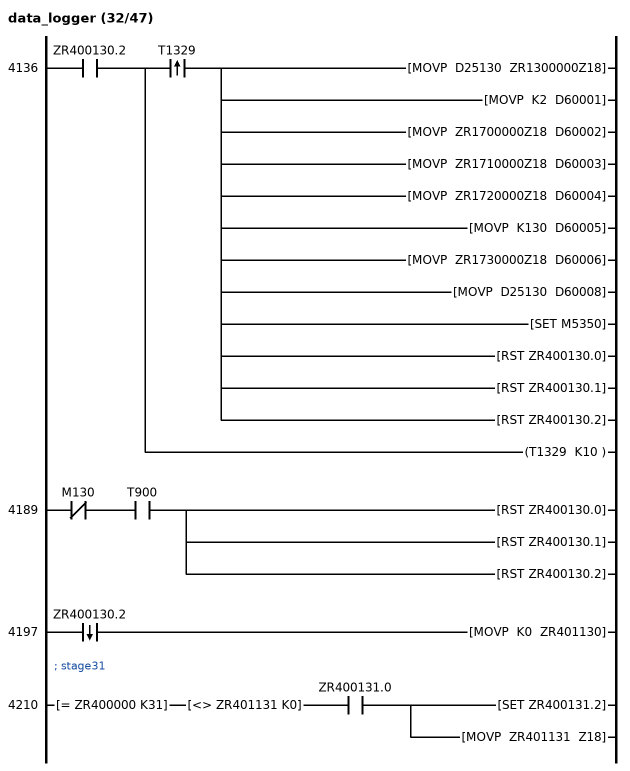
4136  LD      ZR400130.2
      MPS
      ANDP    T1329
      MOVP    D25130 ZR1300000Z18
      MOVP    K2 D60001
      MOVP    ZR1700000Z18 D60002
      MOVP    ZR1710000Z18 D60003
      MOVP    ZR1720000Z18 D60004
      MOVP    K130 D60005
      MOVP    ZR1730000Z18 D60006
      MOVP    D25130 D60008
      SET     M5350
      RST     ZR400130.0
      RST     ZR400130.1
      RST     ZR400130.2
      MPP
      OUT     T1329 K10
4189  LDI     M130
      AND     T900
      RST     ZR400130.0
      RST     ZR400130.1
      RST     ZR400130.2
4197  LDF     ZR400130.2
      MOVP    K0 ZR401130
; stage31
4210  LD=     ZR400000 K31
      AND<>   ZR401131 K0
      AND     ZR400131.0
      SET     ZR400131.2
      MOVP    ZR401131 Z18
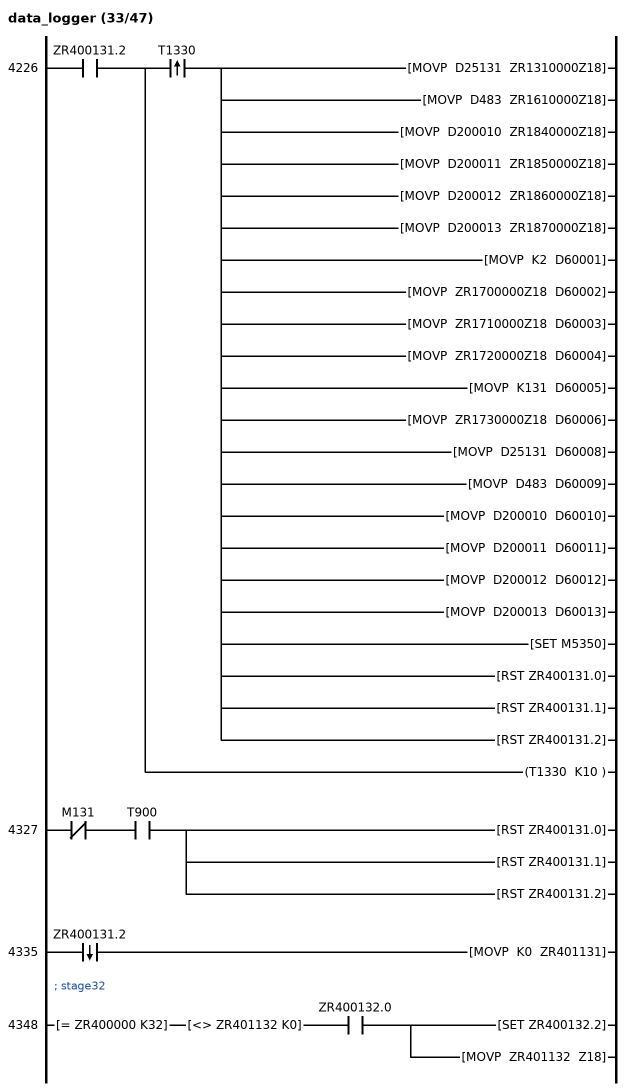
4226  LD      ZR400131.2
      MPS
      ANDP    T1330
      MOVP    D25131 ZR1310000Z18
      MOVP    D483 ZR1610000Z18
      MOVP    D200010 ZR1840000Z18
      MOVP    D200011 ZR1850000Z18
      MOVP    D200012 ZR1860000Z18
      MOVP    D200013 ZR1870000Z18
      MOVP    K2 D60001
      MOVP    ZR1700000Z18 D60002
      MOVP    ZR1710000Z18 D60003
      MOVP    ZR1720000Z18 D60004
      MOVP    K131 D60005
      MOVP    ZR1730000Z18 D60006
      MOVP    D25131 D60008
      MOVP    D483 D60009
      MOVP    D200010 D60010
      MOVP    D200011 D60011
      MOVP    D200012 D60012
      MOVP    D200013 D60013
      SET     M5350
      RST     ZR400131.0
      RST     ZR400131.1
      RST     ZR400131.2
      MPP
      OUT     T1330 K10
4327  LDI     M131
      AND     T900
      RST     ZR400131.0
      RST     ZR400131.1
      RST     ZR400131.2
4335  LDF     ZR400131.2
      MOVP    K0 ZR401131
; stage32
4348  LD=     ZR400000 K32
      AND<>   ZR401132 K0
      AND     ZR400132.0
      SET     ZR400132.2
      MOVP    ZR401132 Z18
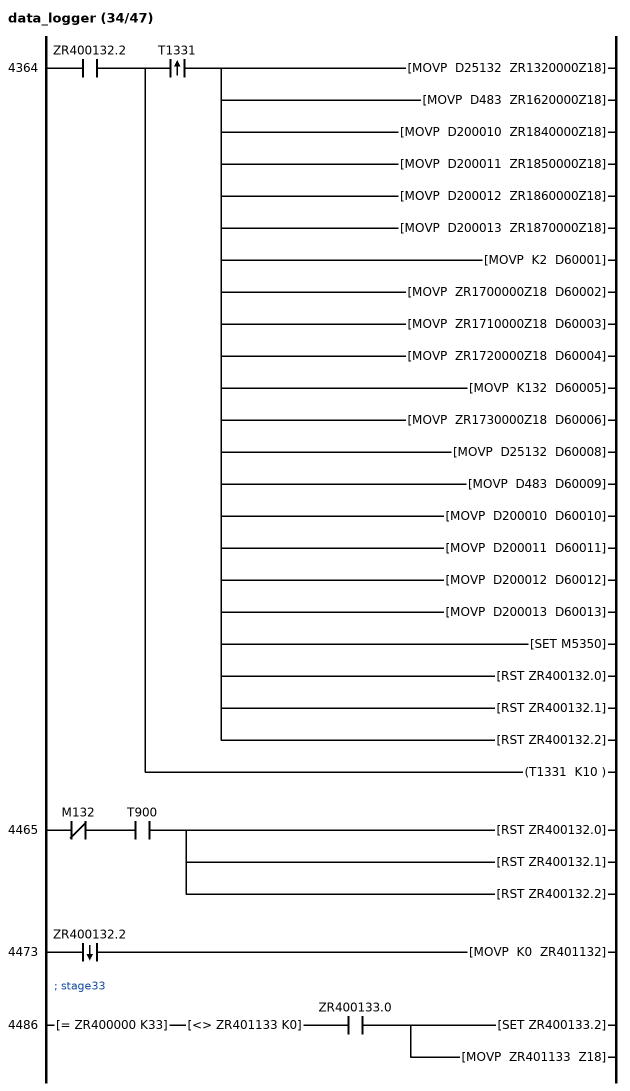
4364  LD      ZR400132.2
      MPS
      ANDP    T1331
      MOVP    D25132 ZR1320000Z18
      MOVP    D483 ZR1620000Z18
      MOVP    D200010 ZR1840000Z18
      MOVP    D200011 ZR1850000Z18
      MOVP    D200012 ZR1860000Z18
      MOVP    D200013 ZR1870000Z18
      MOVP    K2 D60001
      MOVP    ZR1700000Z18 D60002
      MOVP    ZR1710000Z18 D60003
      MOVP    ZR1720000Z18 D60004
      MOVP    K132 D60005
      MOVP    ZR1730000Z18 D60006
      MOVP    D25132 D60008
      MOVP    D483 D60009
      MOVP    D200010 D60010
      MOVP    D200011 D60011
      MOVP    D200012 D60012
      MOVP    D200013 D60013
      SET     M5350
      RST     ZR400132.0
      RST     ZR400132.1
      RST     ZR400132.2
      MPP
      OUT     T1331 K10
4465  LDI     M132
      AND     T900
      RST     ZR400132.0
      RST     ZR400132.1
      RST     ZR400132.2
4473  LDF     ZR400132.2
      MOVP    K0 ZR401132
; stage33
4486  LD=     ZR400000 K33
      AND<>   ZR401133 K0
      AND     ZR400133.0
      SET     ZR400133.2
      MOVP    ZR401133 Z18
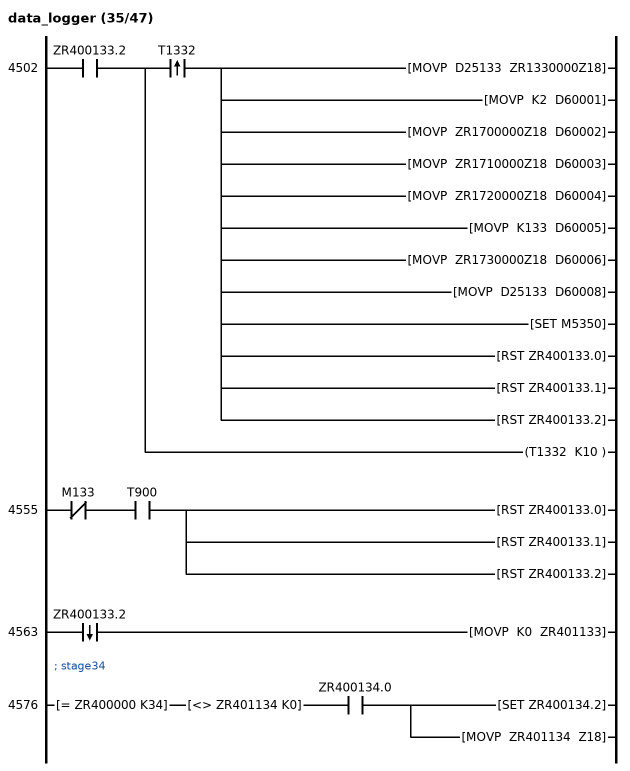
4502  LD      ZR400133.2
      MPS
      ANDP    T1332
      MOVP    D25133 ZR1330000Z18
      MOVP    K2 D60001
      MOVP    ZR1700000Z18 D60002
      MOVP    ZR1710000Z18 D60003
      MOVP    ZR1720000Z18 D60004
      MOVP    K133 D60005
      MOVP    ZR1730000Z18 D60006
      MOVP    D25133 D60008
      SET     M5350
      RST     ZR400133.0
      RST     ZR400133.1
      RST     ZR400133.2
      MPP
      OUT     T1332 K10
4555  LDI     M133
      AND     T900
      RST     ZR400133.0
      RST     ZR400133.1
      RST     ZR400133.2
4563  LDF     ZR400133.2
      MOVP    K0 ZR401133
; stage34
4576  LD=     ZR400000 K34
      AND<>   ZR401134 K0
      AND     ZR400134.0
      SET     ZR400134.2
      MOVP    ZR401134 Z18
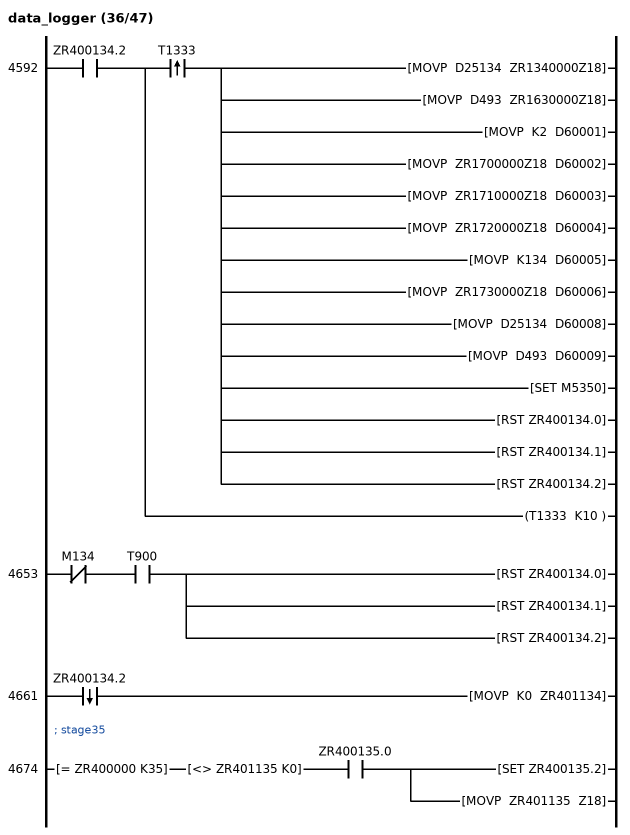
4592  LD      ZR400134.2
      MPS
      ANDP    T1333
      MOVP    D25134 ZR1340000Z18
      MOVP    D493 ZR1630000Z18
      MOVP    K2 D60001
      MOVP    ZR1700000Z18 D60002
      MOVP    ZR1710000Z18 D60003
      MOVP    ZR1720000Z18 D60004
      MOVP    K134 D60005
      MOVP    ZR1730000Z18 D60006
      MOVP    D25134 D60008
      MOVP    D493 D60009
      SET     M5350
      RST     ZR400134.0
      RST     ZR400134.1
      RST     ZR400134.2
      MPP
      OUT     T1333 K10
4653  LDI     M134
      AND     T900
      RST     ZR400134.0
      RST     ZR400134.1
      RST     ZR400134.2
4661  LDF     ZR400134.2
      MOVP    K0 ZR401134
; stage35
4674  LD=     ZR400000 K35
      AND<>   ZR401135 K0
      AND     ZR400135.0
      SET     ZR400135.2
      MOVP    ZR401135 Z18
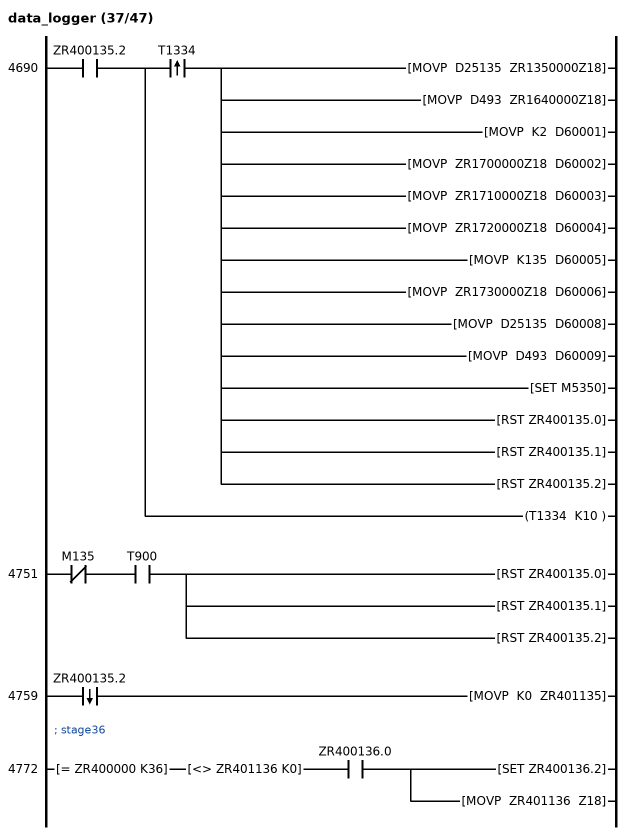
4690  LD      ZR400135.2
      MPS
      ANDP    T1334
      MOVP    D25135 ZR1350000Z18
      MOVP    D493 ZR1640000Z18
      MOVP    K2 D60001
      MOVP    ZR1700000Z18 D60002
      MOVP    ZR1710000Z18 D60003
      MOVP    ZR1720000Z18 D60004
      MOVP    K135 D60005
      MOVP    ZR1730000Z18 D60006
      MOVP    D25135 D60008
      MOVP    D493 D60009
      SET     M5350
      RST     ZR400135.0
      RST     ZR400135.1
      RST     ZR400135.2
      MPP
      OUT     T1334 K10
4751  LDI     M135
      AND     T900
      RST     ZR400135.0
      RST     ZR400135.1
      RST     ZR400135.2
4759  LDF     ZR400135.2
      MOVP    K0 ZR401135
; stage36
4772  LD=     ZR400000 K36
      AND<>   ZR401136 K0
      AND     ZR400136.0
      SET     ZR400136.2
      MOVP    ZR401136 Z18
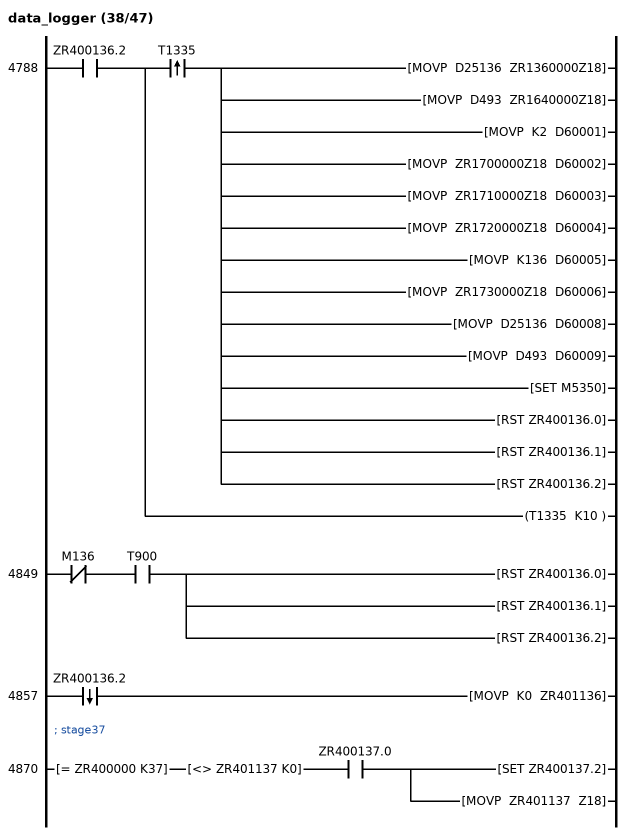
4788  LD      ZR400136.2
      MPS
      ANDP    T1335
      MOVP    D25136 ZR1360000Z18
      MOVP    D493 ZR1640000Z18
      MOVP    K2 D60001
      MOVP    ZR1700000Z18 D60002
      MOVP    ZR1710000Z18 D60003
      MOVP    ZR1720000Z18 D60004
      MOVP    K136 D60005
      MOVP    ZR1730000Z18 D60006
      MOVP    D25136 D60008
      MOVP    D493 D60009
      SET     M5350
      RST     ZR400136.0
      RST     ZR400136.1
      RST     ZR400136.2
      MPP
      OUT     T1335 K10
4849  LDI     M136
      AND     T900
      RST     ZR400136.0
      RST     ZR400136.1
      RST     ZR400136.2
4857  LDF     ZR400136.2
      MOVP    K0 ZR401136
; stage37
4870  LD=     ZR400000 K37
      AND<>   ZR401137 K0
      AND     ZR400137.0
      SET     ZR400137.2
      MOVP    ZR401137 Z18
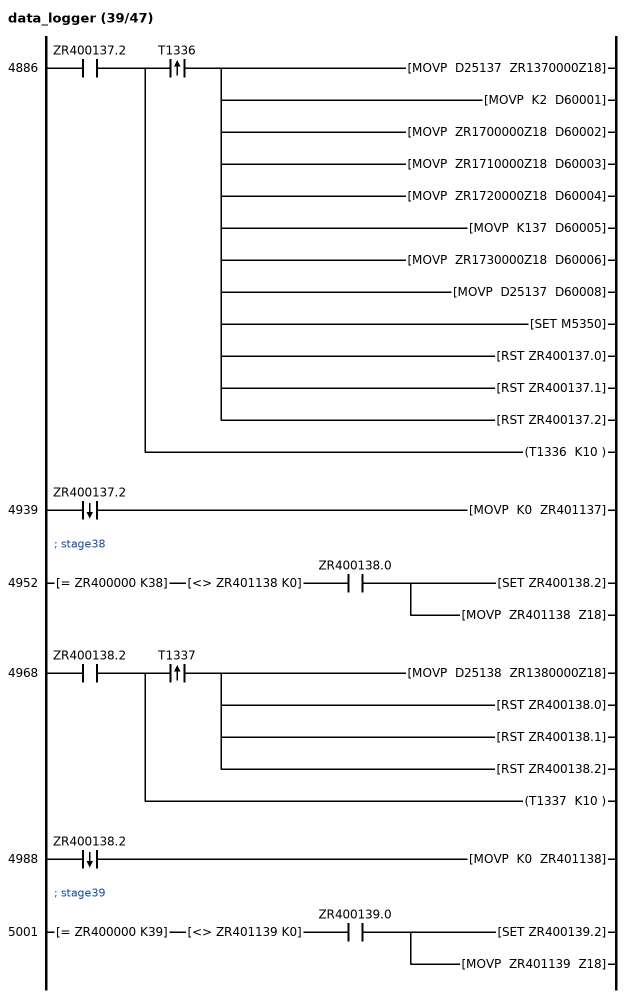
4886  LD      ZR400137.2
      MPS
      ANDP    T1336
      MOVP    D25137 ZR1370000Z18
      MOVP    K2 D60001
      MOVP    ZR1700000Z18 D60002
      MOVP    ZR1710000Z18 D60003
      MOVP    ZR1720000Z18 D60004
      MOVP    K137 D60005
      MOVP    ZR1730000Z18 D60006
      MOVP    D25137 D60008
      SET     M5350
      RST     ZR400137.0
      RST     ZR400137.1
      RST     ZR400137.2
      MPP
      OUT     T1336 K10
4939  LDF     ZR400137.2
      MOVP    K0 ZR401137
; stage38
4952  LD=     ZR400000 K38
      AND<>   ZR401138 K0
      AND     ZR400138.0
      SET     ZR400138.2
      MOVP    ZR401138 Z18
4968  LD      ZR400138.2
      MPS
      ANDP    T1337
      MOVP    D25138 ZR1380000Z18
      RST     ZR400138.0
      RST     ZR400138.1
      RST     ZR400138.2
      MPP
      OUT     T1337 K10
4988  LDF     ZR400138.2
      MOVP    K0 ZR401138
; stage39
5001  LD=     ZR400000 K39
      AND<>   ZR401139 K0
      AND     ZR400139.0
      SET     ZR400139.2
      MOVP    ZR401139 Z18
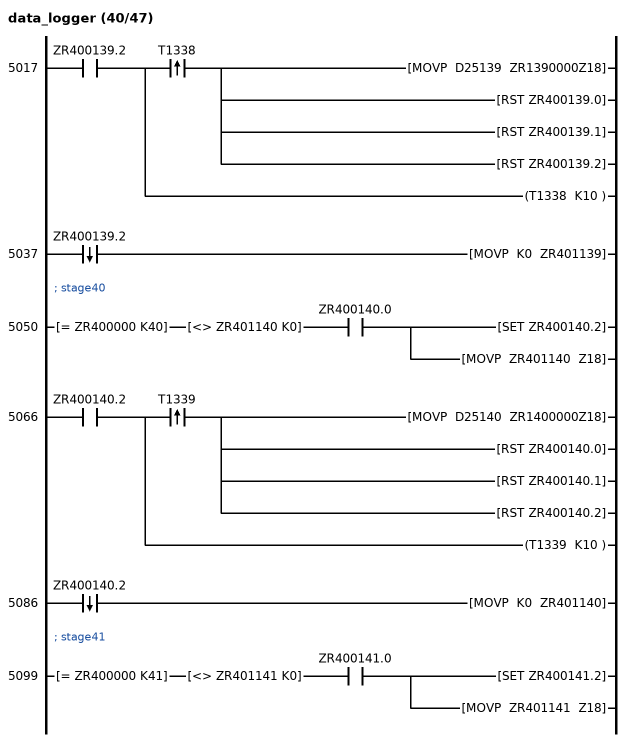
5017  LD      ZR400139.2
      MPS
      ANDP    T1338
      MOVP    D25139 ZR1390000Z18
      RST     ZR400139.0
      RST     ZR400139.1
      RST     ZR400139.2
      MPP
      OUT     T1338 K10
5037  LDF     ZR400139.2
      MOVP    K0 ZR401139
; stage40
5050  LD=     ZR400000 K40
      AND<>   ZR401140 K0
      AND     ZR400140.0
      SET     ZR400140.2
      MOVP    ZR401140 Z18
5066  LD      ZR400140.2
      MPS
      ANDP    T1339
      MOVP    D25140 ZR1400000Z18
      RST     ZR400140.0
      RST     ZR400140.1
      RST     ZR400140.2
      MPP
      OUT     T1339 K10
5086  LDF     ZR400140.2
      MOVP    K0 ZR401140
; stage41
5099  LD=     ZR400000 K41
      AND<>   ZR401141 K0
      AND     ZR400141.0
      SET     ZR400141.2
      MOVP    ZR401141 Z18
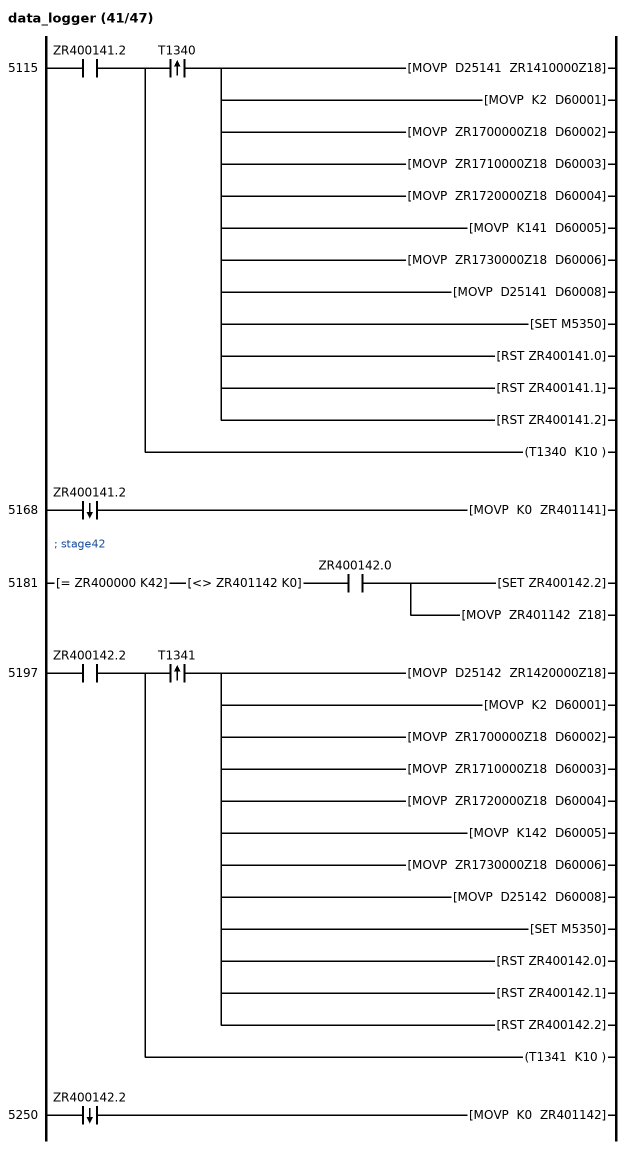
5115  LD      ZR400141.2
      MPS
      ANDP    T1340
      MOVP    D25141 ZR1410000Z18
      MOVP    K2 D60001
      MOVP    ZR1700000Z18 D60002
      MOVP    ZR1710000Z18 D60003
      MOVP    ZR1720000Z18 D60004
      MOVP    K141 D60005
      MOVP    ZR1730000Z18 D60006
      MOVP    D25141 D60008
      SET     M5350
      RST     ZR400141.0
      RST     ZR400141.1
      RST     ZR400141.2
      MPP
      OUT     T1340 K10
5168  LDF     ZR400141.2
      MOVP    K0 ZR401141
; stage42
5181  LD=     ZR400000 K42
      AND<>   ZR401142 K0
      AND     ZR400142.0
      SET     ZR400142.2
      MOVP    ZR401142 Z18
5197  LD      ZR400142.2
      MPS
      ANDP    T1341
      MOVP    D25142 ZR1420000Z18
      MOVP    K2 D60001
      MOVP    ZR1700000Z18 D60002
      MOVP    ZR1710000Z18 D60003
      MOVP    ZR1720000Z18 D60004
      MOVP    K142 D60005
      MOVP    ZR1730000Z18 D60006
      MOVP    D25142 D60008
      SET     M5350
      RST     ZR400142.0
      RST     ZR400142.1
      RST     ZR400142.2
      MPP
      OUT     T1341 K10
5250  LDF     ZR400142.2
      MOVP    K0 ZR401142
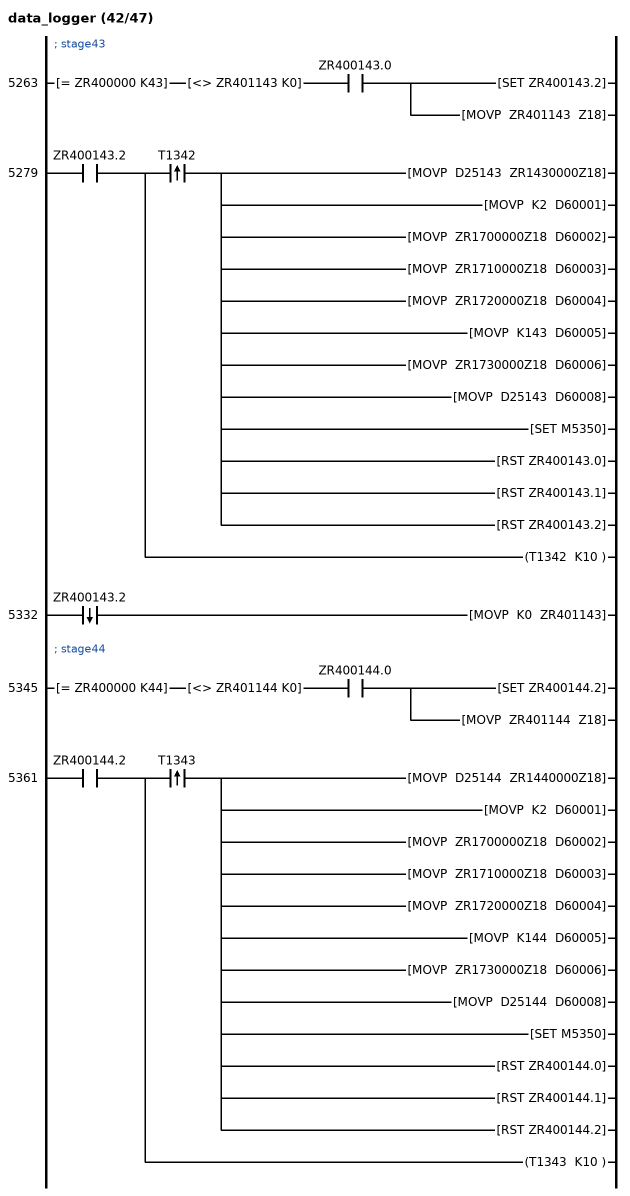
; stage43
5263  LD=     ZR400000 K43
      AND<>   ZR401143 K0
      AND     ZR400143.0
      SET     ZR400143.2
      MOVP    ZR401143 Z18
5279  LD      ZR400143.2
      MPS
      ANDP    T1342
      MOVP    D25143 ZR1430000Z18
      MOVP    K2 D60001
      MOVP    ZR1700000Z18 D60002
      MOVP    ZR1710000Z18 D60003
      MOVP    ZR1720000Z18 D60004
      MOVP    K143 D60005
      MOVP    ZR1730000Z18 D60006
      MOVP    D25143 D60008
      SET     M5350
      RST     ZR400143.0
      RST     ZR400143.1
      RST     ZR400143.2
      MPP
      OUT     T1342 K10
5332  LDF     ZR400143.2
      MOVP    K0 ZR401143
; stage44
5345  LD=     ZR400000 K44
      AND<>   ZR401144 K0
      AND     ZR400144.0
      SET     ZR400144.2
      MOVP    ZR401144 Z18
5361  LD      ZR400144.2
      MPS
      ANDP    T1343
      MOVP    D25144 ZR1440000Z18
      MOVP    K2 D60001
      MOVP    ZR1700000Z18 D60002
      MOVP    ZR1710000Z18 D60003
      MOVP    ZR1720000Z18 D60004
      MOVP    K144 D60005
      MOVP    ZR1730000Z18 D60006
      MOVP    D25144 D60008
      SET     M5350
      RST     ZR400144.0
      RST     ZR400144.1
      RST     ZR400144.2
      MPP
      OUT     T1343 K10
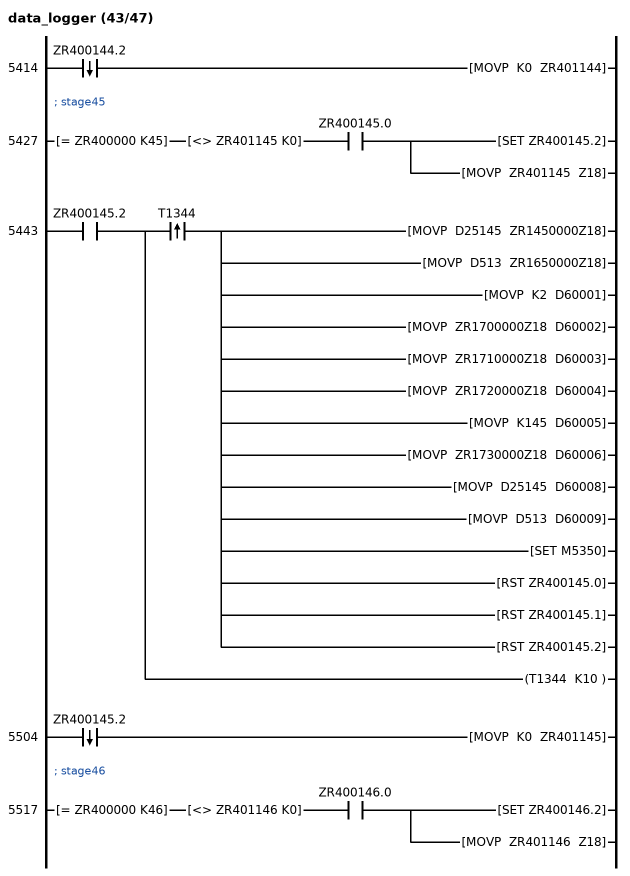
5414  LDF     ZR400144.2
      MOVP    K0 ZR401144
; stage45
5427  LD=     ZR400000 K45
      AND<>   ZR401145 K0
      AND     ZR400145.0
      SET     ZR400145.2
      MOVP    ZR401145 Z18
5443  LD      ZR400145.2
      MPS
      ANDP    T1344
      MOVP    D25145 ZR1450000Z18
      MOVP    D513 ZR1650000Z18
      MOVP    K2 D60001
      MOVP    ZR1700000Z18 D60002
      MOVP    ZR1710000Z18 D60003
      MOVP    ZR1720000Z18 D60004
      MOVP    K145 D60005
      MOVP    ZR1730000Z18 D60006
      MOVP    D25145 D60008
      MOVP    D513 D60009
      SET     M5350
      RST     ZR400145.0
      RST     ZR400145.1
      RST     ZR400145.2
      MPP
      OUT     T1344 K10
5504  LDF     ZR400145.2
      MOVP    K0 ZR401145
; stage46
5517  LD=     ZR400000 K46
      AND<>   ZR401146 K0
      AND     ZR400146.0
      SET     ZR400146.2
      MOVP    ZR401146 Z18
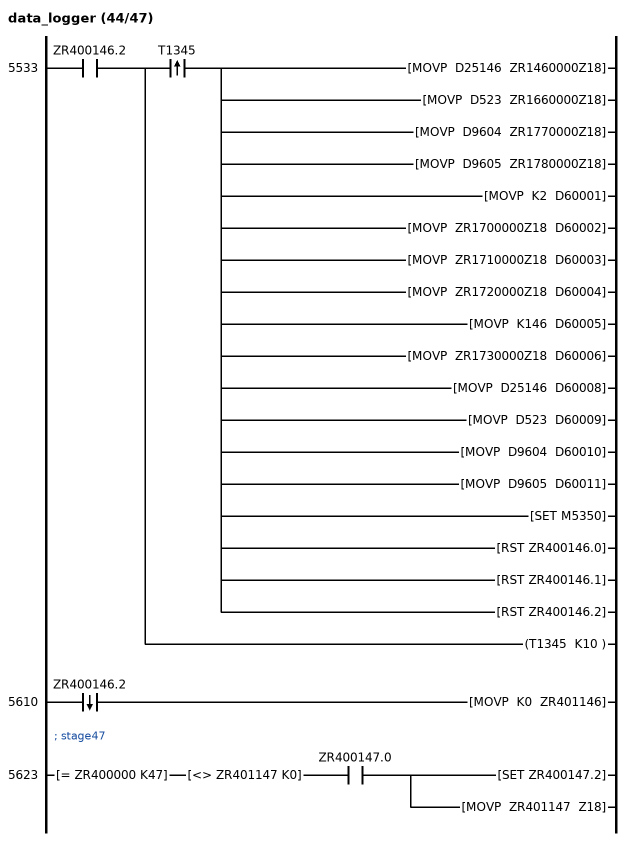
5533  LD      ZR400146.2
      MPS
      ANDP    T1345
      MOVP    D25146 ZR1460000Z18
      MOVP    D523 ZR1660000Z18
      MOVP    D9604 ZR1770000Z18
      MOVP    D9605 ZR1780000Z18
      MOVP    K2 D60001
      MOVP    ZR1700000Z18 D60002
      MOVP    ZR1710000Z18 D60003
      MOVP    ZR1720000Z18 D60004
      MOVP    K146 D60005
      MOVP    ZR1730000Z18 D60006
      MOVP    D25146 D60008
      MOVP    D523 D60009
      MOVP    D9604 D60010
      MOVP    D9605 D60011
      SET     M5350
      RST     ZR400146.0
      RST     ZR400146.1
      RST     ZR400146.2
      MPP
      OUT     T1345 K10
5610  LDF     ZR400146.2
      MOVP    K0 ZR401146
; stage47
5623  LD=     ZR400000 K47
      AND<>   ZR401147 K0
      AND     ZR400147.0
      SET     ZR400147.2
      MOVP    ZR401147 Z18
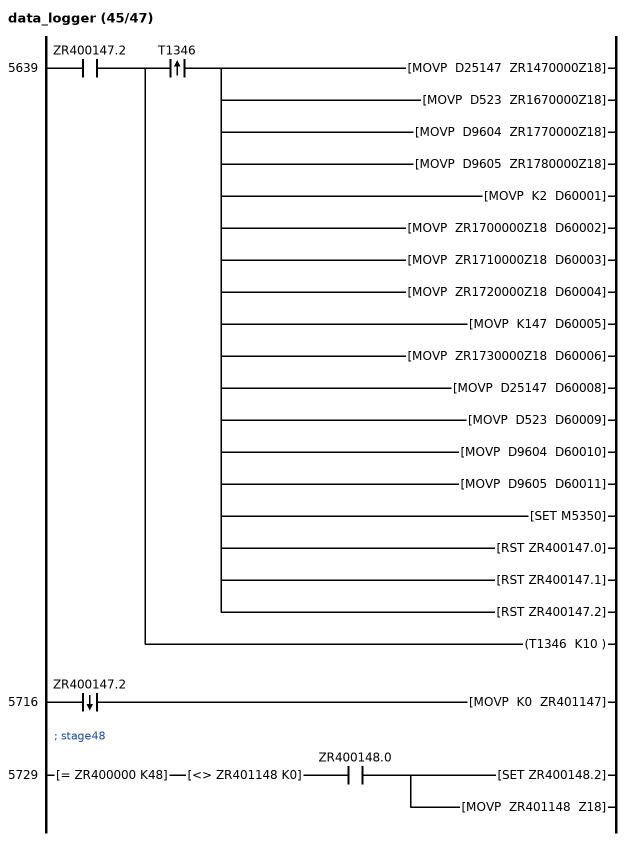
5639  LD      ZR400147.2
      MPS
      ANDP    T1346
      MOVP    D25147 ZR1470000Z18
      MOVP    D523 ZR1670000Z18
      MOVP    D9604 ZR1770000Z18
      MOVP    D9605 ZR1780000Z18
      MOVP    K2 D60001
      MOVP    ZR1700000Z18 D60002
      MOVP    ZR1710000Z18 D60003
      MOVP    ZR1720000Z18 D60004
      MOVP    K147 D60005
      MOVP    ZR1730000Z18 D60006
      MOVP    D25147 D60008
      MOVP    D523 D60009
      MOVP    D9604 D60010
      MOVP    D9605 D60011
      SET     M5350
      RST     ZR400147.0
      RST     ZR400147.1
      RST     ZR400147.2
      MPP
      OUT     T1346 K10
5716  LDF     ZR400147.2
      MOVP    K0 ZR401147
; stage48
5729  LD=     ZR400000 K48
      AND<>   ZR401148 K0
      AND     ZR400148.0
      SET     ZR400148.2
      MOVP    ZR401148 Z18
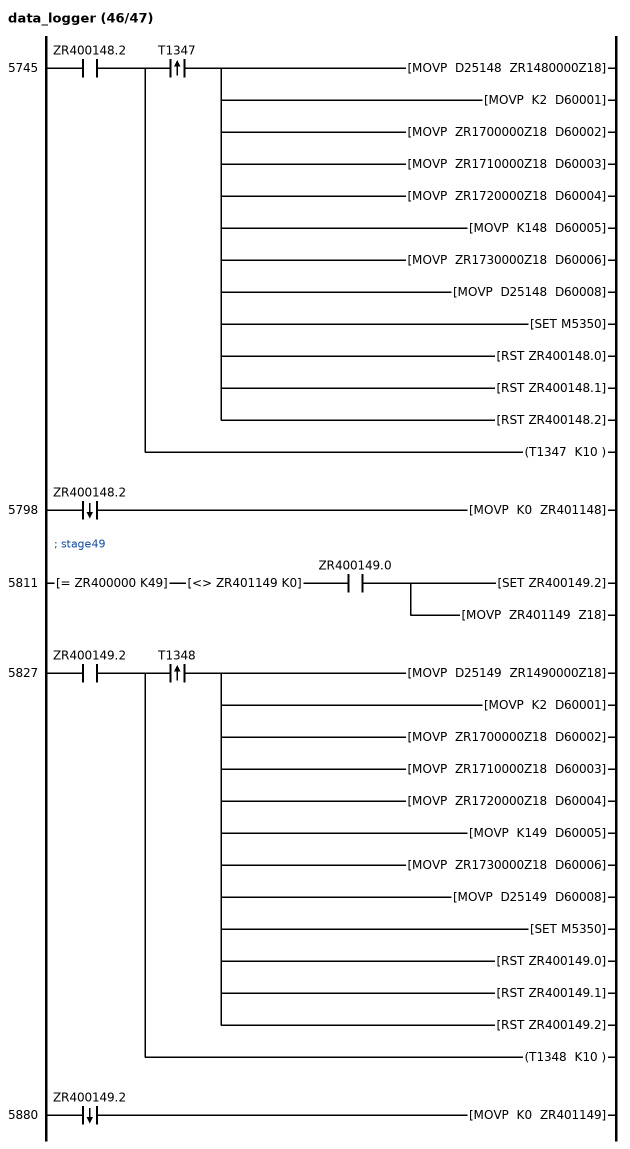
5745  LD      ZR400148.2
      MPS
      ANDP    T1347
      MOVP    D25148 ZR1480000Z18
      MOVP    K2 D60001
      MOVP    ZR1700000Z18 D60002
      MOVP    ZR1710000Z18 D60003
      MOVP    ZR1720000Z18 D60004
      MOVP    K148 D60005
      MOVP    ZR1730000Z18 D60006
      MOVP    D25148 D60008
      SET     M5350
      RST     ZR400148.0
      RST     ZR400148.1
      RST     ZR400148.2
      MPP
      OUT     T1347 K10
5798  LDF     ZR400148.2
      MOVP    K0 ZR401148
; stage49
5811  LD=     ZR400000 K49
      AND<>   ZR401149 K0
      AND     ZR400149.0
      SET     ZR400149.2
      MOVP    ZR401149 Z18
5827  LD      ZR400149.2
      MPS
      ANDP    T1348
      MOVP    D25149 ZR1490000Z18
      MOVP    K2 D60001
      MOVP    ZR1700000Z18 D60002
      MOVP    ZR1710000Z18 D60003
      MOVP    ZR1720000Z18 D60004
      MOVP    K149 D60005
      MOVP    ZR1730000Z18 D60006
      MOVP    D25149 D60008
      SET     M5350
      RST     ZR400149.0
      RST     ZR400149.1
      RST     ZR400149.2
      MPP
      OUT     T1348 K10
5880  LDF     ZR400149.2
      MOVP    K0 ZR401149
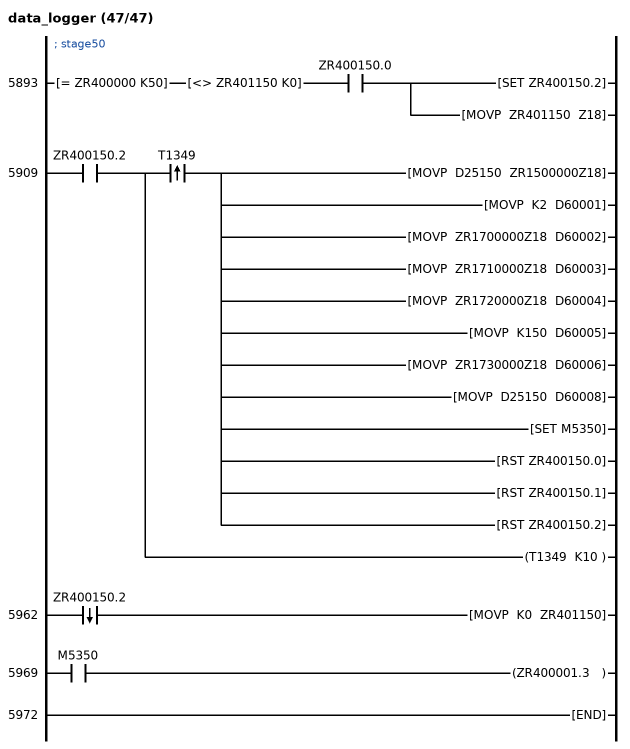
; stage50
5893  LD=     ZR400000 K50
      AND<>   ZR401150 K0
      AND     ZR400150.0
      SET     ZR400150.2
      MOVP    ZR401150 Z18
5909  LD      ZR400150.2
      MPS
      ANDP    T1349
      MOVP    D25150 ZR1500000Z18
      MOVP    K2 D60001
      MOVP    ZR1700000Z18 D60002
      MOVP    ZR1710000Z18 D60003
      MOVP    ZR1720000Z18 D60004
      MOVP    K150 D60005
      MOVP    ZR1730000Z18 D60006
      MOVP    D25150 D60008
      SET     M5350
      RST     ZR400150.0
      RST     ZR400150.1
      RST     ZR400150.2
      MPP
      OUT     T1349 K10
5962  LDF     ZR400150.2
      MOVP    K0 ZR401150
5969  LD      M5350
      OUT     ZR400001.3
5972  END
END_PROGRAM

PROGRAM data_logger_R
VAR
  __IST_b7c0c6d72a974ae8 : I+ST_b7c0c6d72a974ae8;
  __IST_f649ea45d16546a8 : I+ST_f649ea45d16546a8;
END_VAR
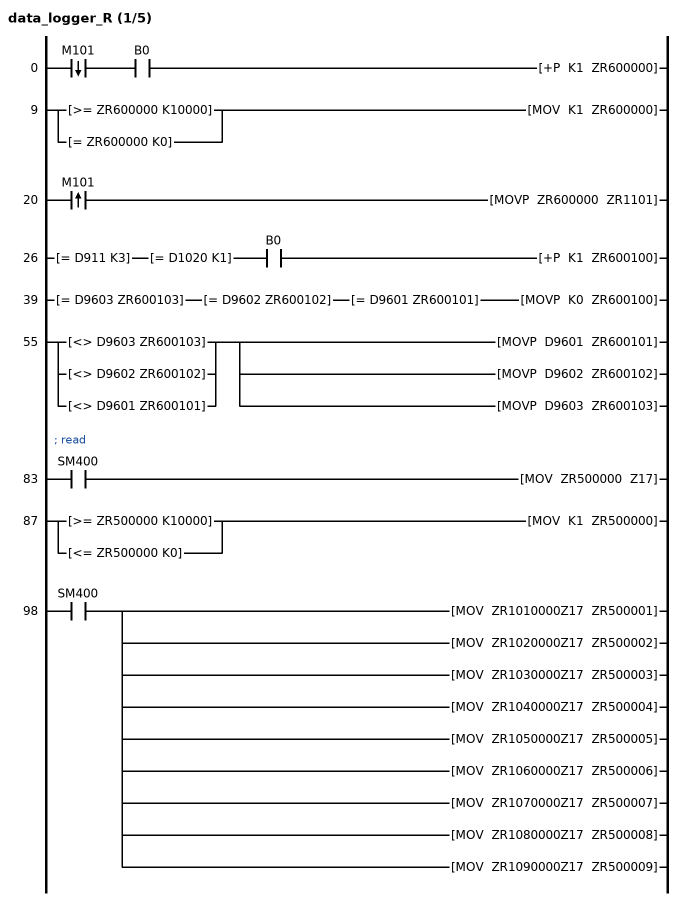
0     LDF     M101
      AND     B0
      +P      K1 ZR600000
9     LD>=    ZR600000 K10000
      OR=     ZR600000 K0
      MOV     K1 ZR600000
20    LDP     M101
      MOVP    ZR600000 ZR1101
26    LD=     D911 K3
      AND=    D1020 K1
      AND     B0
      +P      K1 ZR600100
39    LD=     D9603 ZR600103
      AND=    D9602 ZR600102
      AND=    D9601 ZR600101
      MOVP    K0 ZR600100
55    LD<>    D9603 ZR600103
      OR<>    D9602 ZR600102
      OR<>    D9601 ZR600101
      MOVP    D9601 ZR600101
      MOVP    D9602 ZR600102
      MOVP    D9603 ZR600103
; read
83    LD      SM400
      MOV     ZR500000 Z17
87    LD>=    ZR500000 K10000
      OR<=    ZR500000 K0
      MOV     K1 ZR500000
98    LD      SM400
      MOV     ZR1010000Z17 ZR500001
      MOV     ZR1020000Z17 ZR500002
      MOV     ZR1030000Z17 ZR500003
      MOV     ZR1040000Z17 ZR500004
      MOV     ZR1050000Z17 ZR500005
      MOV     ZR1060000Z17 ZR500006
      MOV     ZR1070000Z17 ZR500007
      MOV     ZR1080000Z17 ZR500008
      MOV     ZR1090000Z17 ZR500009
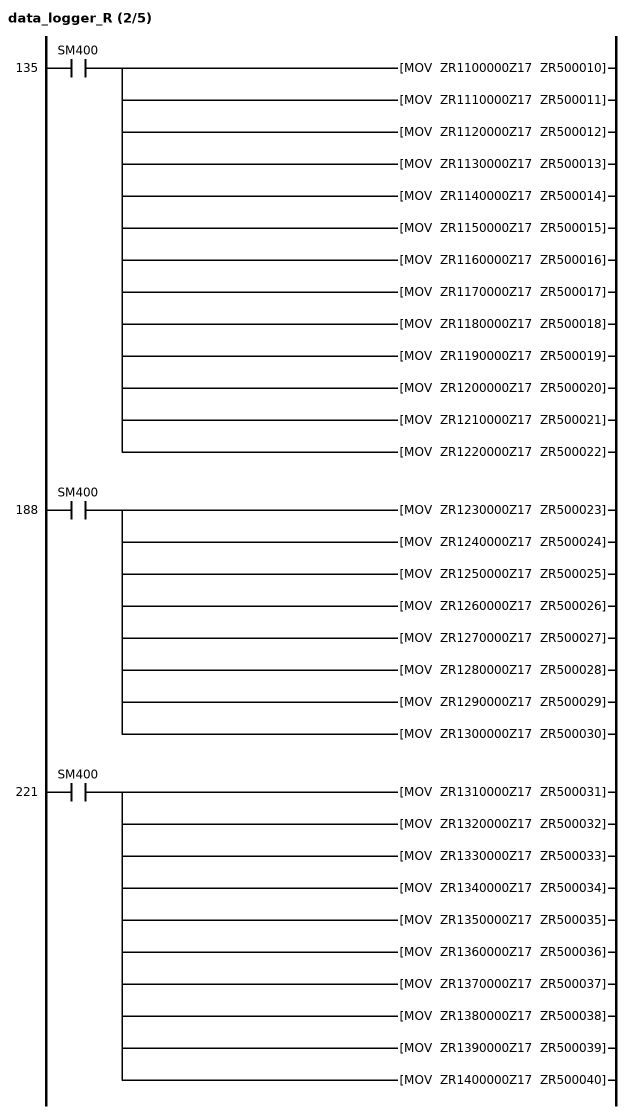
135   LD      SM400
      MOV     ZR1100000Z17 ZR500010
      MOV     ZR1110000Z17 ZR500011
      MOV     ZR1120000Z17 ZR500012
      MOV     ZR1130000Z17 ZR500013
      MOV     ZR1140000Z17 ZR500014
      MOV     ZR1150000Z17 ZR500015
      MOV     ZR1160000Z17 ZR500016
      MOV     ZR1170000Z17 ZR500017
      MOV     ZR1180000Z17 ZR500018
      MOV     ZR1190000Z17 ZR500019
      MOV     ZR1200000Z17 ZR500020
      MOV     ZR1210000Z17 ZR500021
      MOV     ZR1220000Z17 ZR500022
188   LD      SM400
      MOV     ZR1230000Z17 ZR500023
      MOV     ZR1240000Z17 ZR500024
      MOV     ZR1250000Z17 ZR500025
      MOV     ZR1260000Z17 ZR500026
      MOV     ZR1270000Z17 ZR500027
      MOV     ZR1280000Z17 ZR500028
      MOV     ZR1290000Z17 ZR500029
      MOV     ZR1300000Z17 ZR500030
221   LD      SM400
      MOV     ZR1310000Z17 ZR500031
      MOV     ZR1320000Z17 ZR500032
      MOV     ZR1330000Z17 ZR500033
      MOV     ZR1340000Z17 ZR500034
      MOV     ZR1350000Z17 ZR500035
      MOV     ZR1360000Z17 ZR500036
      MOV     ZR1370000Z17 ZR500037
      MOV     ZR1380000Z17 ZR500038
      MOV     ZR1390000Z17 ZR500039
      MOV     ZR1400000Z17 ZR500040
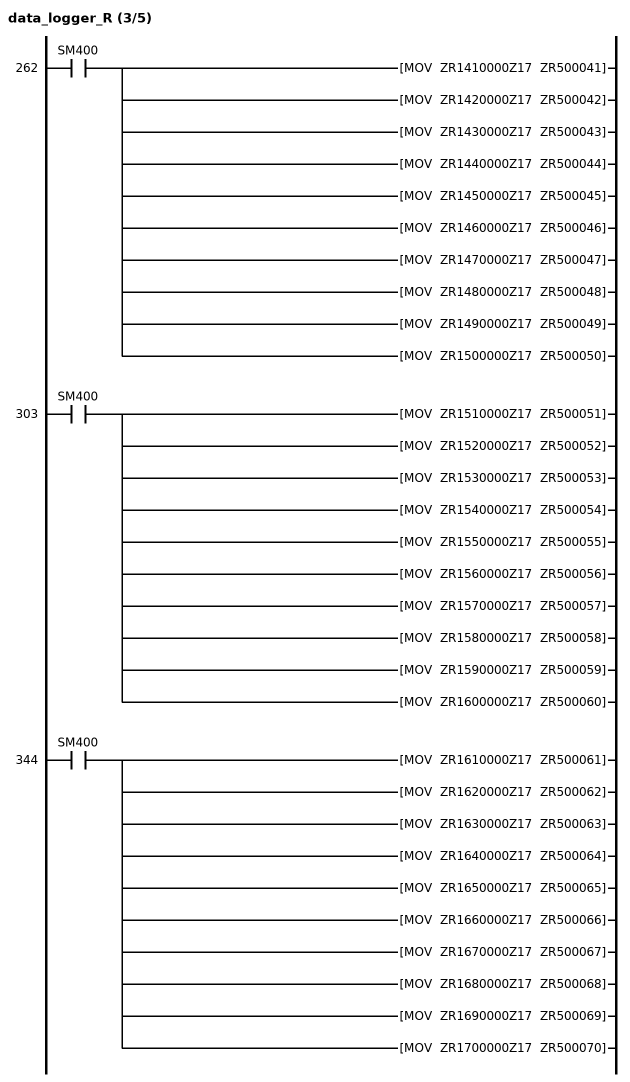
262   LD      SM400
      MOV     ZR1410000Z17 ZR500041
      MOV     ZR1420000Z17 ZR500042
      MOV     ZR1430000Z17 ZR500043
      MOV     ZR1440000Z17 ZR500044
      MOV     ZR1450000Z17 ZR500045
      MOV     ZR1460000Z17 ZR500046
      MOV     ZR1470000Z17 ZR500047
      MOV     ZR1480000Z17 ZR500048
      MOV     ZR1490000Z17 ZR500049
      MOV     ZR1500000Z17 ZR500050
303   LD      SM400
      MOV     ZR1510000Z17 ZR500051
      MOV     ZR1520000Z17 ZR500052
      MOV     ZR1530000Z17 ZR500053
      MOV     ZR1540000Z17 ZR500054
      MOV     ZR1550000Z17 ZR500055
      MOV     ZR1560000Z17 ZR500056
      MOV     ZR1570000Z17 ZR500057
      MOV     ZR1580000Z17 ZR500058
      MOV     ZR1590000Z17 ZR500059
      MOV     ZR1600000Z17 ZR500060
344   LD      SM400
      MOV     ZR1610000Z17 ZR500061
      MOV     ZR1620000Z17 ZR500062
      MOV     ZR1630000Z17 ZR500063
      MOV     ZR1640000Z17 ZR500064
      MOV     ZR1650000Z17 ZR500065
      MOV     ZR1660000Z17 ZR500066
      MOV     ZR1670000Z17 ZR500067
      MOV     ZR1680000Z17 ZR500068
      MOV     ZR1690000Z17 ZR500069
      MOV     ZR1700000Z17 ZR500070
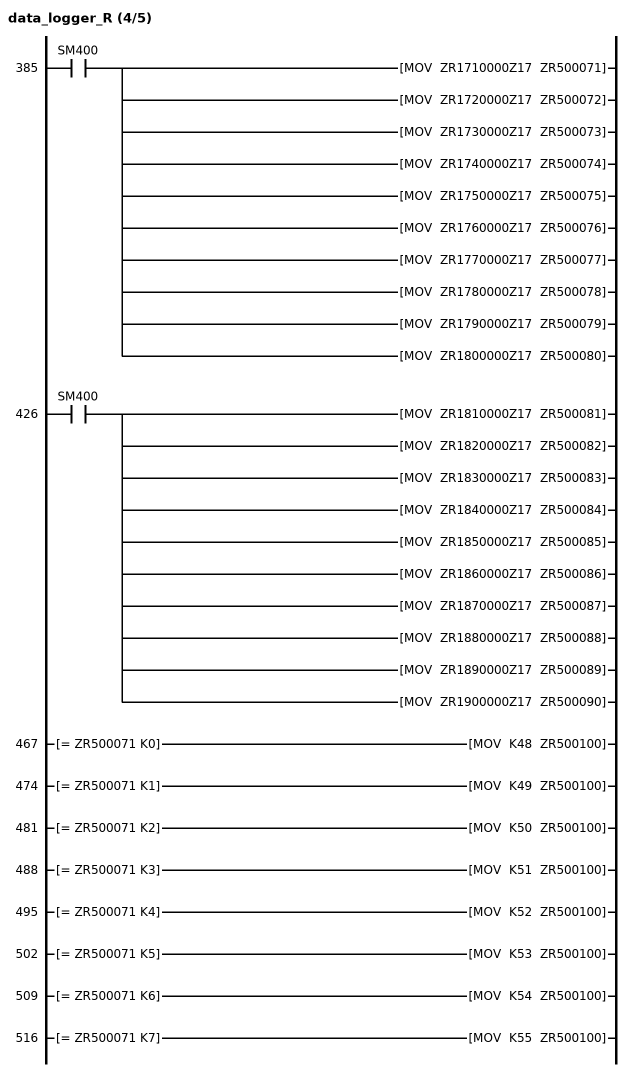
385   LD      SM400
      MOV     ZR1710000Z17 ZR500071
      MOV     ZR1720000Z17 ZR500072
      MOV     ZR1730000Z17 ZR500073
      MOV     ZR1740000Z17 ZR500074
      MOV     ZR1750000Z17 ZR500075
      MOV     ZR1760000Z17 ZR500076
      MOV     ZR1770000Z17 ZR500077
      MOV     ZR1780000Z17 ZR500078
      MOV     ZR1790000Z17 ZR500079
      MOV     ZR1800000Z17 ZR500080
426   LD      SM400
      MOV     ZR1810000Z17 ZR500081
      MOV     ZR1820000Z17 ZR500082
      MOV     ZR1830000Z17 ZR500083
      MOV     ZR1840000Z17 ZR500084
      MOV     ZR1850000Z17 ZR500085
      MOV     ZR1860000Z17 ZR500086
      MOV     ZR1870000Z17 ZR500087
      MOV     ZR1880000Z17 ZR500088
      MOV     ZR1890000Z17 ZR500089
      MOV     ZR1900000Z17 ZR500090
467   LD=     ZR500071 K0
      MOV     K48 ZR500100
474   LD=     ZR500071 K1
      MOV     K49 ZR500100
481   LD=     ZR500071 K2
      MOV     K50 ZR500100
488   LD=     ZR500071 K3
      MOV     K51 ZR500100
495   LD=     ZR500071 K4
      MOV     K52 ZR500100
502   LD=     ZR500071 K5
      MOV     K53 ZR500100
509   LD=     ZR500071 K6
      MOV     K54 ZR500100
516   LD=     ZR500071 K7
      MOV     K55 ZR500100
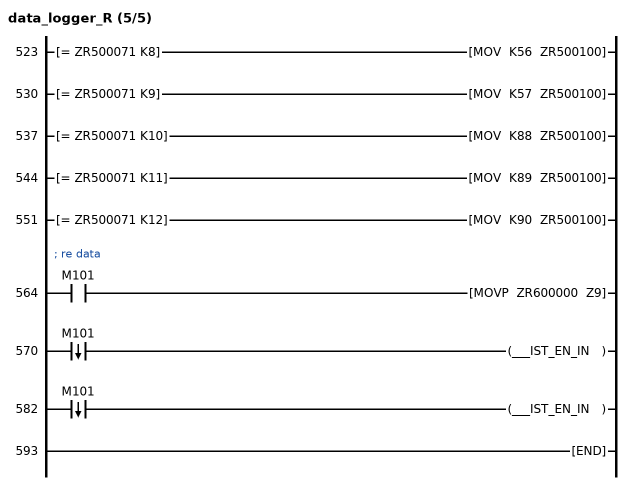
523   LD=     ZR500071 K8
      MOV     K56 ZR500100
530   LD=     ZR500071 K9
      MOV     K57 ZR500100
537   LD=     ZR500071 K10
      MOV     K88 ZR500100
544   LD=     ZR500071 K11
      MOV     K89 ZR500100
551   LD=     ZR500071 K12
      MOV     K90 ZR500100
; re data
564   LD      M101
      MOVP    ZR600000 Z9
; FB BLK START I+ST_b7c0c6d72a974ae8(__IST_b7c0c6d72a974ae8)
570   LDF     M101
      OUT     ___IST_EN_IN
; FB START
; FB_NAME I+ST_b7c0c6d72a974ae8
; INSTANCE_NAME __IST_b7c0c6d72a974ae8
; FB IN_B:__IST_EN_IN
; FB OUT___IST_EN_OUT:B
; FB END
; FB BLK END
; FB BLK START I+ST_f649ea45d16546a8(__IST_f649ea45d16546a8)
582   LDF     M101
      OUT     ___IST_EN_IN
; FB START
; FB_NAME I+ST_f649ea45d16546a8
; INSTANCE_NAME __IST_f649ea45d16546a8
; FB IN_B:__IST_EN_IN
; FB OUT___IST_EN_OUT:B
; FB END
; FB BLK END
593   END
END_PROGRAM

PROGRAM DBV3
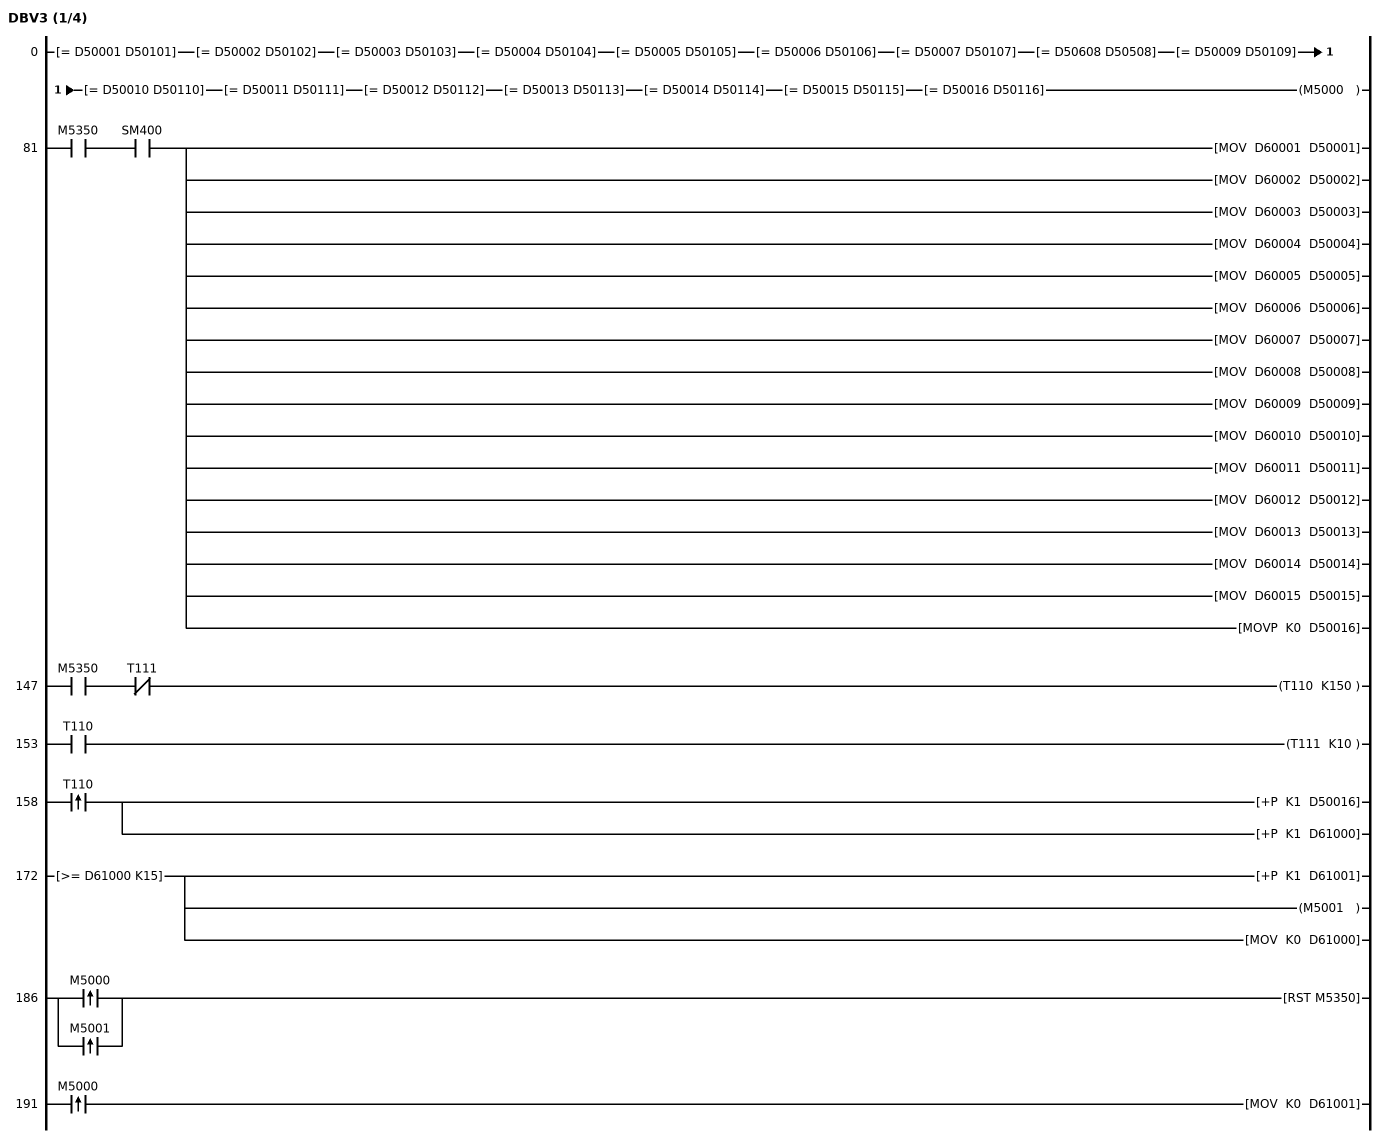
0     LD=     D50001 D50101
      AND=    D50002 D50102
      AND=    D50003 D50103
      AND=    D50004 D50104
      AND=    D50005 D50105
      AND=    D50006 D50106
      AND=    D50007 D50107
      AND=    D50608 D50508
      AND=    D50009 D50109
      AND=    D50010 D50110
      AND=    D50011 D50111
      AND=    D50012 D50112
      AND=    D50013 D50113
      AND=    D50014 D50114
      AND=    D50015 D50115
      AND=    D50016 D50116
      OUT     M5000
81    LD      M5350
      AND     SM400
      MOV     D60001 D50001
      MOV     D60002 D50002
      MOV     D60003 D50003
      MOV     D60004 D50004
      MOV     D60005 D50005
      MOV     D60006 D50006
      MOV     D60007 D50007
      MOV     D60008 D50008
      MOV     D60009 D50009
      MOV     D60010 D50010
      MOV     D60011 D50011
      MOV     D60012 D50012
      MOV     D60013 D50013
      MOV     D60014 D50014
      MOV     D60015 D50015
      MOVP    K0 D50016
147   LD      M5350
      ANI     T111
      OUT     T110 K150
153   LD      T110
      OUT     T111 K10
158   LDP     T110
      +P      K1 D50016
      +P      K1 D61000
172   LD>=    D61000 K15
      +P      K1 D61001
      OUT     M5001
      MOV     K0 D61000
186   LDP     M5000
      ORP     M5001
      RST     M5350
191   LDP     M5000
      MOV     K0 D61001
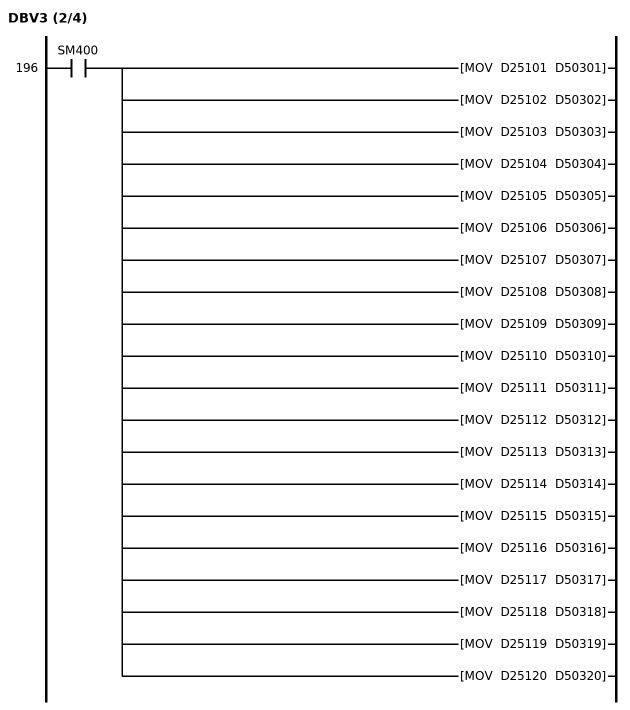
196   LD      SM400
      MOV     D25101 D50301
      MOV     D25102 D50302
      MOV     D25103 D50303
      MOV     D25104 D50304
      MOV     D25105 D50305
      MOV     D25106 D50306
      MOV     D25107 D50307
      MOV     D25108 D50308
      MOV     D25109 D50309
      MOV     D25110 D50310
      MOV     D25111 D50311
      MOV     D25112 D50312
      MOV     D25113 D50313
      MOV     D25114 D50314
      MOV     D25115 D50315
      MOV     D25116 D50316
      MOV     D25117 D50317
      MOV     D25118 D50318
      MOV     D25119 D50319
      MOV     D25120 D50320
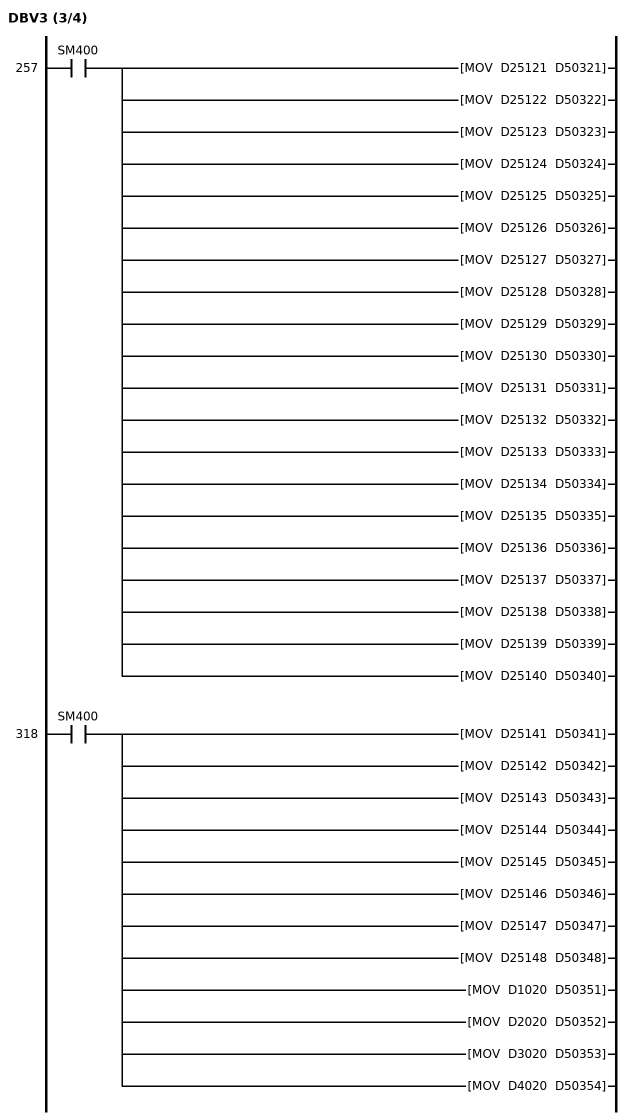
257   LD      SM400
      MOV     D25121 D50321
      MOV     D25122 D50322
      MOV     D25123 D50323
      MOV     D25124 D50324
      MOV     D25125 D50325
      MOV     D25126 D50326
      MOV     D25127 D50327
      MOV     D25128 D50328
      MOV     D25129 D50329
      MOV     D25130 D50330
      MOV     D25131 D50331
      MOV     D25132 D50332
      MOV     D25133 D50333
      MOV     D25134 D50334
      MOV     D25135 D50335
      MOV     D25136 D50336
      MOV     D25137 D50337
      MOV     D25138 D50338
      MOV     D25139 D50339
      MOV     D25140 D50340
318   LD      SM400
      MOV     D25141 D50341
      MOV     D25142 D50342
      MOV     D25143 D50343
      MOV     D25144 D50344
      MOV     D25145 D50345
      MOV     D25146 D50346
      MOV     D25147 D50347
      MOV     D25148 D50348
      MOV     D1020 D50351
      MOV     D2020 D50352
      MOV     D3020 D50353
      MOV     D4020 D50354
